(* IEC 61131-3 sources: TIA2AX/tests/test_projects/_expected/PLC_1, 6 files *)

(* ---- HwInputs.st ---- *)
TYPE
	HwInputs : STRUCT
		IO_device_1_DI_8x24VDC_BA_1 AT %B0 : BYTE;
	END_STRUCT;
END_TYPE

(* ---- HwOutputs.st ---- *)
TYPE
	HwOutputs : STRUCT
	END_STRUCT;
END_TYPE

(* ---- PlcInputs.st ---- *)
TYPE
	PlcInputs : STRUCT
		IO_device_1_DI_8x24VDC_BA_1 : BYTE;
	END_STRUCT;
END_TYPE

(* ---- PlcOutputs.st ---- *)
TYPE
	PlcOutputs : STRUCT
	END_STRUCT;
END_TYPE

(* ---- CopyInputs.st ---- *)
FUNCTION CopyInputs
	VAR_EXTERNAL
		HwInputs : HwInputs;
		PlcInputs : PlcInputs;
	END_VAR
	PlcInputs.IO_device_1_DI_8x24VDC_BA_1 := HwInputs.IO_device_1_DI_8x24VDC_BA_1;
END_FUNCTION

(* ---- CopyOutputs.st ---- *)
FUNCTION CopyOutputs
	VAR_EXTERNAL
		HwOutputs : HwOutputs;
		PlcOutputs : PlcOutputs;
	END_VAR
END_FUNCTION
